// TIA Portal V16 export
// export: Created 2021-04-11T09:51:30.9739273Z, ExportSetting WithDefaults, DisplayName Totally Integrated Automation Portal, DisplayVersion V16, DisplayName TIA Portal Version Control Interface, DisplayVersion V16, DisplayName TIA Portal Openness, DisplayVersion V16, DisplayName STEP 7 Professional, DisplayVersion V16, DisplayName STEP 7 Safety, DisplayVersion V16, DisplayName WinCC Unified SCADA Engineering System, DisplayVersion V16
TYPE "addedVibro"
// stored: IsFailsafeCompliant false
   STRUCT
      manStartVibroTable : Array[0..2] of Bool;   // запуск вибростола в ручном режиме
      manValueVibro : Int;   // величина вибрации в ручном режиме
      stateVibroTable : Array[0..2] of Bool;
   END_STRUCT;
END_TYPE
